# EPICS substitutions: bts_vacuumApp/Db/bts_vac_tmc.substitutions
file bts_vac_tmc.template {
  pattern
    {PORT}
    {"BTS_VAC_ADS"}
}
